// TIA Portal project "3PhaseMotor" (V18)

(* hardware
DEVICE "S7-1200 station_1"  S7-1200 Station
   slot 0: "Rack_0"  S7-1200 Rack  Rack  V1.0
   slot 1: "PLC_1"  CPU 1211C DC/DC/DC  6ES7 211-1AE40-0XB0  V4.6
*)

// ===== PLC "PLC_1"  CPU 1211C DC/DC/DC =====

VAR_GLOBAL   // PLC tag table "Default tag table"
   "start" AT %I0.0 : Bool;
   "stop" AT %I0.1 : Bool;
   "Motor1" AT %Q0.0 : Bool;
   "Motor2" AT %Q0.1 : Bool;
   "Tag_1" AT %M0.0 : Bool;
   "Tag_2" AT %M0.1 : Bool;
   "Tag_3" AT %M0.2 : Bool;
   "Tag_4" AT %M0.3 : Bool;
   "Tag_5" AT %M0.4 : Bool;
END_VAR

// folder: System blocks/Program resources

DATA_BLOCK "IEC_Timer_0_DB"   // DB1
{ S7_Optimized_Access := 'TRUE' }
AUTHOR : Simatic
FAMILY : IEC
NAME : IEC_TMR
VERSION : 1.0
// stored: InstanceOfName IEC_TIMER
"IEC_TIMER"
BEGIN
END_DATA_BLOCK

DATA_BLOCK "IEC_Timer_0_DB_1"   // DB2
{ S7_Optimized_Access := 'TRUE' }
AUTHOR : Simatic
FAMILY : IEC
NAME : IEC_TMR
VERSION : 1.0
// stored: InstanceOfName IEC_TIMER
"IEC_TIMER"
BEGIN
END_DATA_BLOCK

DATA_BLOCK "IEC_Timer_0_DB_2"   // DB3
{ S7_Optimized_Access := 'TRUE' }
AUTHOR : Simatic
FAMILY : IEC
NAME : IEC_TMR
VERSION : 1.0
// stored: InstanceOfName IEC_TIMER
"IEC_TIMER"
BEGIN
END_DATA_BLOCK

DATA_BLOCK "IEC_Timer_0_DB_3"   // DB4
{ S7_Optimized_Access := 'TRUE' }
AUTHOR : Simatic
FAMILY : IEC
NAME : IEC_TMR
VERSION : 1.0
// stored: InstanceOfName IEC_TIMER
"IEC_TIMER"
BEGIN
END_DATA_BLOCK

// folder: (top level)

ORGANIZATION_BLOCK "Main"   // OB1, LAD, ProgramCycle
TITLE = "Main Program Sweep (Cycle)"
{ S7_Optimized_Access := 'TRUE' }
VERSION : 0.1
   VAR_INPUT
      Initial_Call : Bool;   // Initial call of this OB
      Remanence : Bool;   // =True, if remanent data are available
   END_VAR
   VAR_TEMP   // added for the SCL form of the ladder/FBD networks
      _w1 : Bool;
      _w2 : Bool;
   END_VAR
BEGIN

REGION Network 1
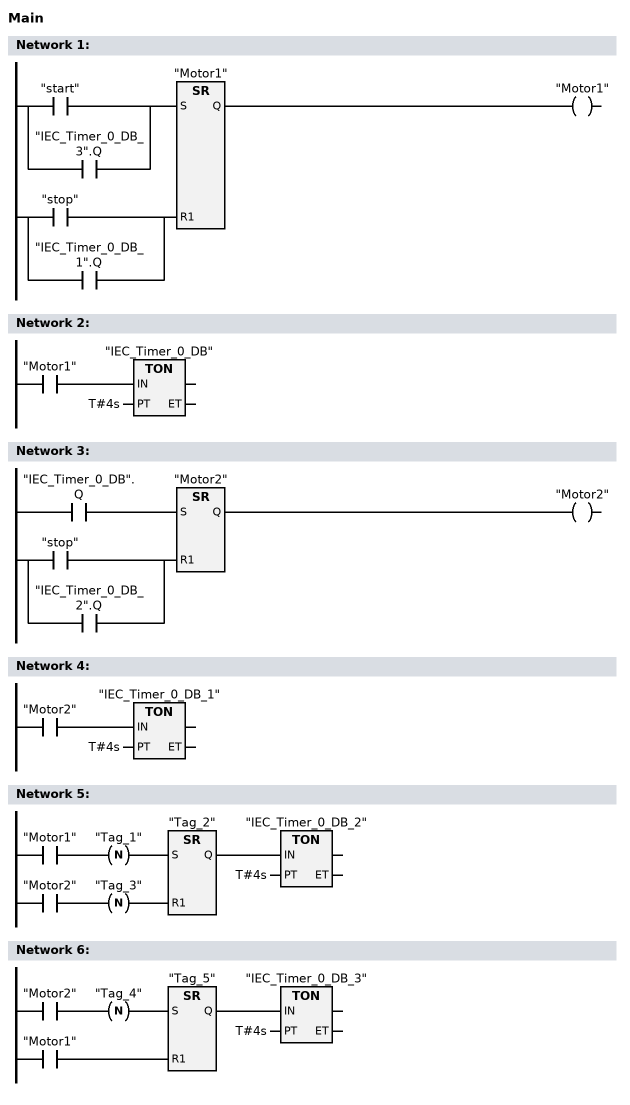
   RUNG wire#powerrail
      Contact( "start" )
      wire#w1
      S_SR(operand := "Motor1", r1 := wire#w2)
      Coil( "Motor1" )
   END_RUNG
   RUNG wire#powerrail
      Contact( "IEC_Timer_0_DB_3".Q )
   END_RUNG wire#w1
   RUNG wire#powerrail
      Contact( "stop" )
   END_RUNG wire#w2
   RUNG wire#powerrail
      Contact( "IEC_Timer_0_DB_1".Q )
   END_RUNG wire#w2
   // the same network as SCL:
   IF "start" OR "IEC_Timer_0_DB_3".Q THEN
       "Motor1" := TRUE;   // SR flip-flop
   END_IF;
   IF "stop" OR "IEC_Timer_0_DB_1".Q THEN "Motor1" := FALSE; END_IF;
   "Motor1" := "Motor1";
END_REGION

REGION Network 2
   "IEC_Timer_0_DB".TON(IN := "Motor1", PT := T#4s);
END_REGION

REGION Network 3
   RUNG wire#powerrail
      Contact( "IEC_Timer_0_DB".Q )
      S_SR(operand := "Motor2", r1 := wire#w1)
      Coil( "Motor2" )
   END_RUNG
   RUNG wire#powerrail
      Contact( "stop" )
   END_RUNG wire#w1
   RUNG wire#powerrail
      Contact( "IEC_Timer_0_DB_2".Q )
   END_RUNG wire#w1
   // the same network as SCL:
   IF "IEC_Timer_0_DB".Q THEN
       "Motor2" := TRUE;   // SR flip-flop
   END_IF;
   IF "stop" OR "IEC_Timer_0_DB_2".Q THEN "Motor2" := FALSE; END_IF;
   "Motor2" := "Motor2";
END_REGION

REGION Network 4
   "IEC_Timer_0_DB_1".TON(IN := "Motor2", PT := T#4s);
END_REGION

REGION Network 5
   #_w1 := NOT "Motor1" AND "Tag_1";   // falling edge
   "Tag_1" := "Motor1";
   #_w2 := NOT "Motor2" AND "Tag_3";   // falling edge
   "Tag_3" := "Motor2";
   IF #_w1 THEN
       "Tag_2" := TRUE;   // SR flip-flop
   END_IF;
   IF #_w2 THEN "Tag_2" := FALSE; END_IF;
   "IEC_Timer_0_DB_2".TON(IN := "Tag_2", PT := T#4s);
END_REGION

REGION Network 6
   #_w1 := NOT "Motor2" AND "Tag_4";   // falling edge
   "Tag_4" := "Motor2";
   IF #_w1 THEN
       "Tag_5" := TRUE;   // SR flip-flop
   END_IF;
   IF "Motor1" THEN "Tag_5" := FALSE; END_IF;
   "IEC_Timer_0_DB_3".TON(IN := "Tag_5", PT := T#4s);
END_REGION
END_ORGANIZATION_BLOCK